{attribute 'GeneratedUsingTerminal: EK1100-0000-0018'}
{attribute addProperty BoxType "EK1100-0000-0018"}
{attribute addProperty Id "Beckhoff_EQ2xxxEK1122Beckhoff_EQ2xxxEK1122_A2ADAD55247"}
{attribute addProperty CRC "3444957817"}
{attribute addProperty Size "247"}
TYPE Beckhoff_EQ2xxx_CD55E279 EXTENDS EK1100_AB5A9467 :
STRUCT
	{attribute addProperty Name "Beckhoff_EQ2xxxEK1122"}
	{attribute addProperty PreviousPort "Beckhoff EQ2xxx : B"}
	Beckhoff_EQ2xxxEK1122 : Beckhoff_EQ2xxxEK1122_A2ADAD55;
END_STRUCT
END_TYPE

(* stored: Version 1.2.0.0, ProductVersion 3.1.4024.9
   DUT Beckhoff_EQ2xxx_CD55E279: Id {db72cf82-320c-4593-9cda-ccb7a5a61343} *)
